FUNCTION_BLOCK FB_HMI_CONTROL_UNITS EXTENDS FB_HMI_COMPONENT
VAR_INPUT
END_VAR
VAR_OUTPUT
END_VAR
VAR
END_VAR

END_FUNCTION_BLOCK

(* stored: Version 1.1.0.1, ProductVersion 3.1.4024.14
   POU FB_HMI_CONTROL_UNITS: Id {fc25dc12-d416-4c28-9188-36c497c6941a}, SpecialFunc None *)
